FUNCTION Fun_Counter : INT
VAR_INPUT
	i_count_in 			: INT; 
END_VAR
VAR
	i_countUp 			: INT := 1;
END_VAR

Fun_Counter := i_count_in + i_countUp;

END_FUNCTION

(* stored: Version 1.1.0.1, ProductVersion 3.1.4024.9
   POU Fun_Counter: Id {6a0e17bb-5c4b-477e-925e-b889edc4f185}, SpecialFunc None *)
